{attribute clr [Container(Layout.Stack)]}
{attribute clr [Group(Layout.Scroll)]}
TYPE CU00xProcessData EXTENDS TcoCore.TcoStruct :
STRUCT
	BoltPresenceInspector : TcoInspectors.TcoDigitalInspector(THISSTRUCT);
END_STRUCT
END_TYPE

(* stored: Version 1.1.0.1, ProductVersion 3.1.4024.9
   DUT CU00xProcessData: Id {3cde27d5-efc5-4d61-b268-7d32d11d85fc} *)
